PROGRAM MAIN
VAR
	hr				:	HRESULT;
	
	fbCamera		:	FB_VN_SimpleCameraControl;
	eState			:	ETcVnCameraState;
	
	ipImageIn		:	ITcVnImage;
	ipImageInDisp	:	ITcVnDisplayableImage;
	
	ipImageRes		:	ITcVnImage;
	ipImageResDisp	:	ITcVnDisplayableImage;
	
	// Pharma-Code
	ipCodeDecodedList 	:	ITcVnContainer;
	ipCodeContourList	:	ITcVnContainer;
	sCodeAsString		: 	STRING(255);
	aCodeContour		:	ARRAY[0..3] OF TcVnPoint2_DINT;

	// Watchdog
	hrWD				:	HRESULT;
	tStop				:	DINT	:= 5000;
	tRest				:	DINT;
	
	// Output
	sText				:	STRING;
	
	// Color
	aColorRed			:	TcVnVector4_LREAL := [255, 0, 0];
END_VAR

//Disclaimer

//THIS publication contains statements about the suitability OF our products FOR certain 
//areas OF application. These statements are based on typical features OF our products. 
//The examples shown in THIS publication are FOR demonstration purposes only. The 
//information provided herein should NOT be regarded as specific operation characteristics. 
//It is incumbent on the customer TO check AND decide whether a product is suitable FOR use 
//in a particular application. We DO NOT give ANY warranty that the source code which is 
//made available with this publication is complete or accurate. 

//THE SAMPLE CODE CONTAINED IN THIS PUBLICATION IS PROVIDED “AS IS” WITHOUT WARRANTY OF ANY 
//KIND, EITHER EXPRESSED, IMPLIED OR STATUTORY, INCLUDING WITHOUT LIMITATION, ANY WARRANTY 
//WITH RESPECT TO NON-INFRINGEMENT, FREEDOM FROM PROPRIETARY RIGHTS OF THIRD PARTIES OR 
//FITNESS FOR ANY PARTICULAR PURPOSE. 

//THIS publication may be changed FROM TIME TO TIME without prior notice. No liability 
//is assumed FOR errors AND/OR omissions. Our products are described in detail in our 
//data sheets AND documentations. Product-specific warnings AND cautions must be observed. 
//FOR the latest version OF our data sheets AND documentations visit our website 
//(www.beckhoff.de). 
 
//© Beckhoff Automation GmbH & Co. KG, March 2020

//The reproduction, distribution AND utilization OF THIS document as well as the 
//communication OF its contents TO others without express authorization is prohibited. 
//Offenders will be held liable FOR the payment OF damages. All rights reserved in the 
//event of the grant of a patent, utility model or design.

//-----------------------------------------------------------------------------------------

// SAMPLE - Pharma-Code Reading
// =================================

// Steps To Do:
// ------------
// 1. Add the sample images to the FileSource1

eState := fbCamera.GetState();

CASE eState OF
	
TCVN_CS_INITIAL, TCVN_CS_INITIALIZING, TCVN_CS_INITIALIZED, TCVN_CS_OPENING, TCVN_CS_OPENED, TCVN_CS_STARTACQUISITION:
	hr := fbCamera.StartAcquisition();
	
TCVN_CS_ACQUIRING:

	hr := fbCamera.GetCurrentImage(ipImageIn);

	IF SUCCEEDED(hr) AND ipImageIn <> 0 THEN

		// Create Result Image
		hr := F_VN_ConvertColorSpace(ipImageIn, ipImageRes, TCVN_CST_Gray_TO_RGB, hr);
	
		// Execute the Pharma Code Reading Function monitored by the Watchdog-Function 
		// --------------------------------------------------------------------------
		hrWD := F_VN_StartRelWatchdog(tStop, S_OK);
			hr := F_VN_ReadPharmaCodeExp(
									ipSrcImage		:= ipImageIn, 
									ipDecodedData	:= ipCodeDecodedList, 
									ipContours		:= ipCodeContourList, 
									nCodeNumber		:= 1,
									nMinBarNumber	:= 4, 
									hrPrev			:= hr);
		hrWD := F_VN_StopWatchdog(hrWD, tRest => tRest);

		// Check if the function was executed successfully 
		IF hr = S_OK THEN
			// Export Code into String
			hr := F_VN_ExportSubContainer_String(ipCodeDecodedList, 0, sCodeAsString, 255, hr);
			
			// Write Code into Result Image
			sText := CONCAT('Code: ', sCodeAsString);
			hr := F_VN_PutTextExp(sText, ipImageRes, 25, 50, ETcVnFontType.TCVN_FT_HERSHEY_PLAIN, 3, aColorRed,2, TCVN_LT_4_CONNECTED, FALSE, hr);
			
			// Draw Code Contour into Result Image
			hr := F_VN_DrawContours(ipCodeContourList, 0, ipImageRes, aColorRed, 3, hr);
			hr := F_VN_ExportSubContainer(ipCodeContourList, 0, ADR(aCodeContour), SIZEOF(aCodeContour), hr);	
		ELSE			
			// Write HRESULT into Result Image
			sText := CONCAT('Returncode ', DINT_TO_STRING(hr));
			hr := F_VN_PutTextExp(sText, ipImageRes, 25, 50, ETcVnFontType.TCVN_FT_HERSHEY_PLAIN, 3, aColorRed,2, TCVN_LT_4_CONNECTED, FALSE, hr);
		END_IF
			
		// Write Code Reading proceeded time into Result Image
		sText := CONCAT(CONCAT('Time: ', DINT_TO_STRING(tStop - tRest)), 'us');
		hr := F_VN_PutTextExp(sText, ipImageRes, 25, 100, ETcVnFontType.TCVN_FT_HERSHEY_PLAIN, 3, aColorRed,2, TCVN_LT_4_CONNECTED, FALSE, hr);
				
		// Display Input Image
		hr := F_VN_TransformIntoDisplayableImage(ipImageIn, ipImageInDisp, hr);
		
		// Disply Result Image
		hr := F_VN_TransformIntoDisplayableImage(ipImageRes, ipImageResDisp, hr);
		
	END_IF

TCVN_CS_ERROR:
	hr := fbCamera.Reset();
	
END_CASE

END_PROGRAM

(* stored: Version 1.1.0.1, ProductVersion 3.1.4024.6
   POU MAIN: Id {37a20a90-f645-4306-a374-ca86c1ba0459}, SpecialFunc None *)
